# B&R Automation Studio project DuctLines (part 16)

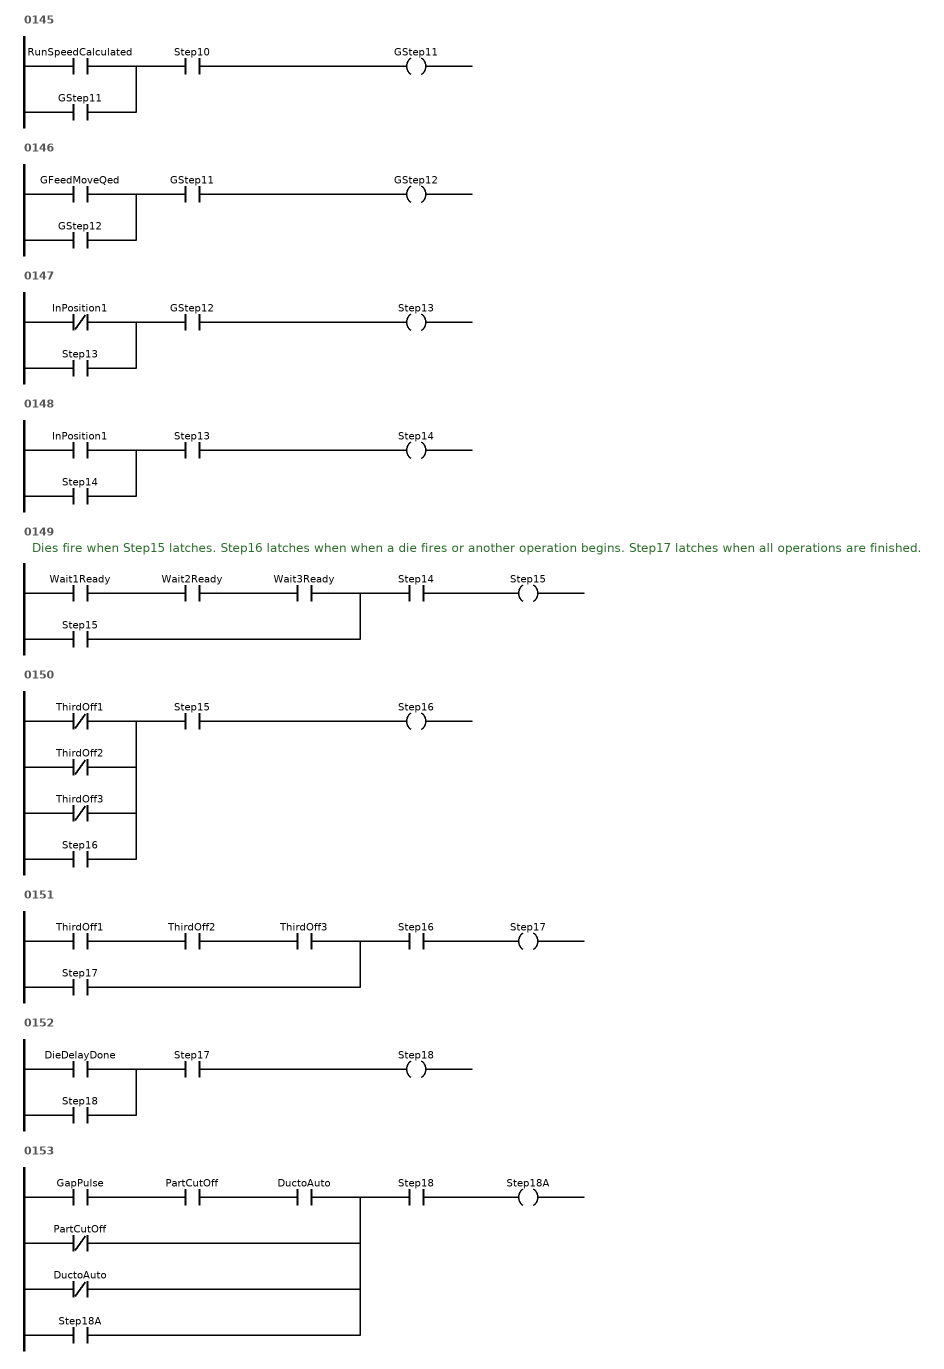
[picture p282: ladder Cyclic.ld]
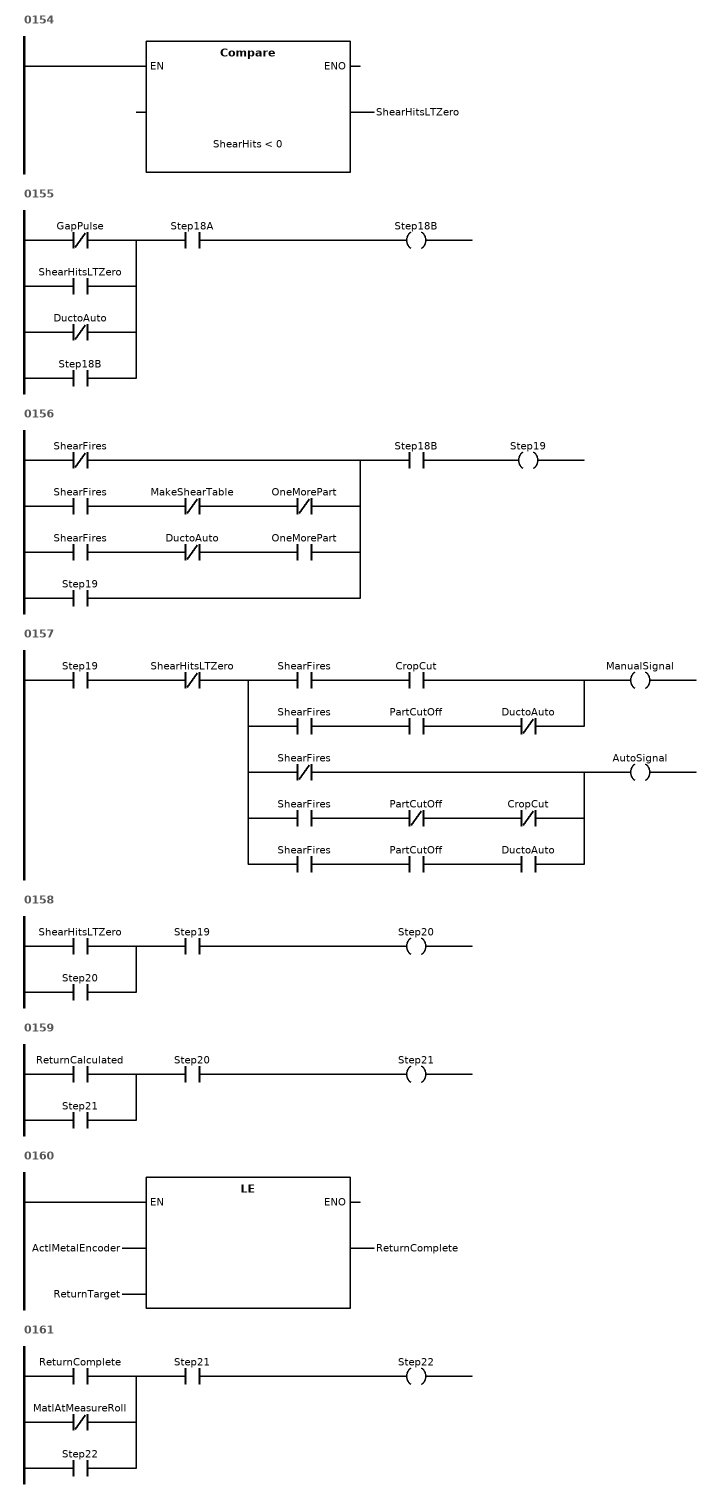
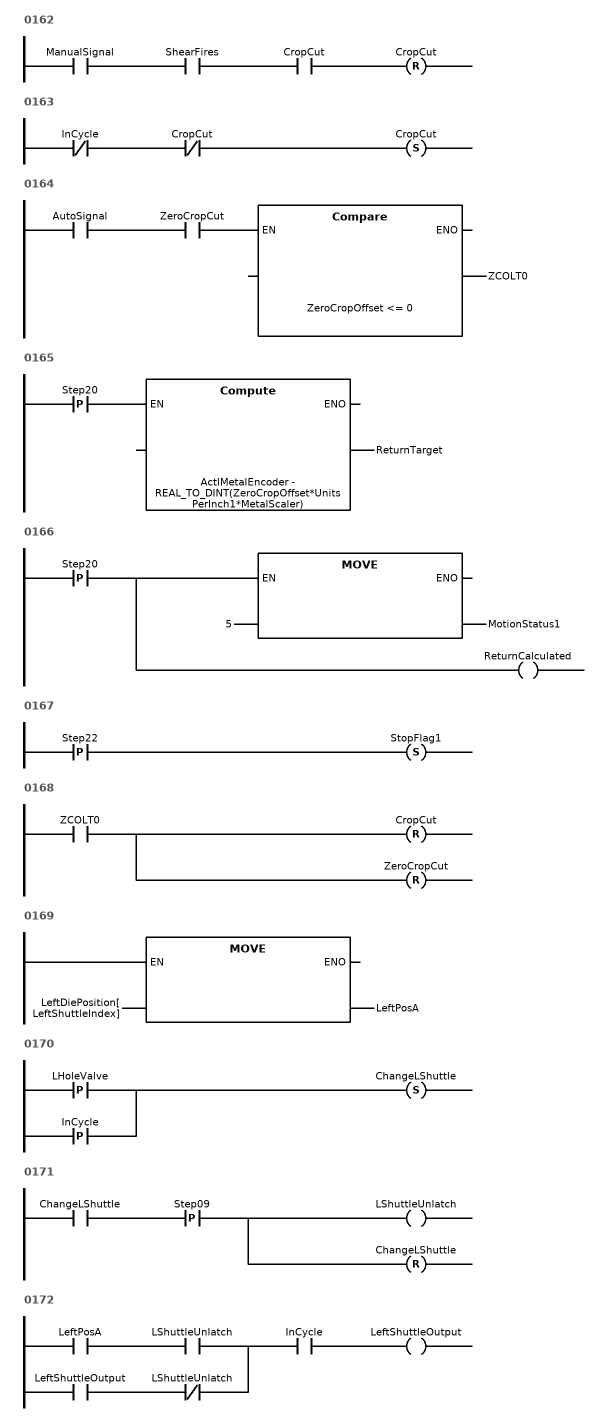
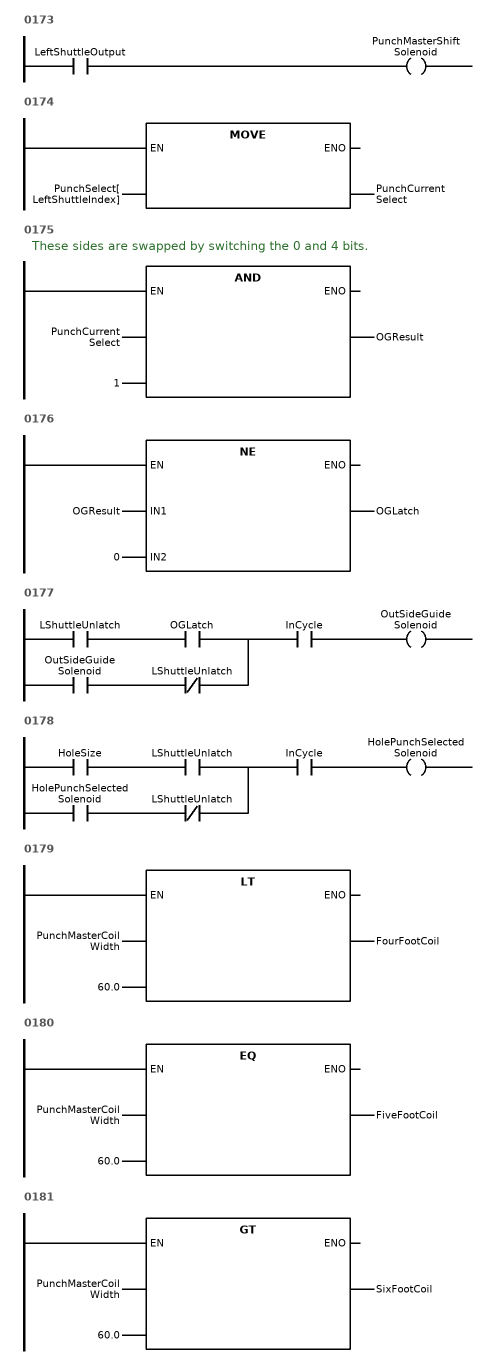
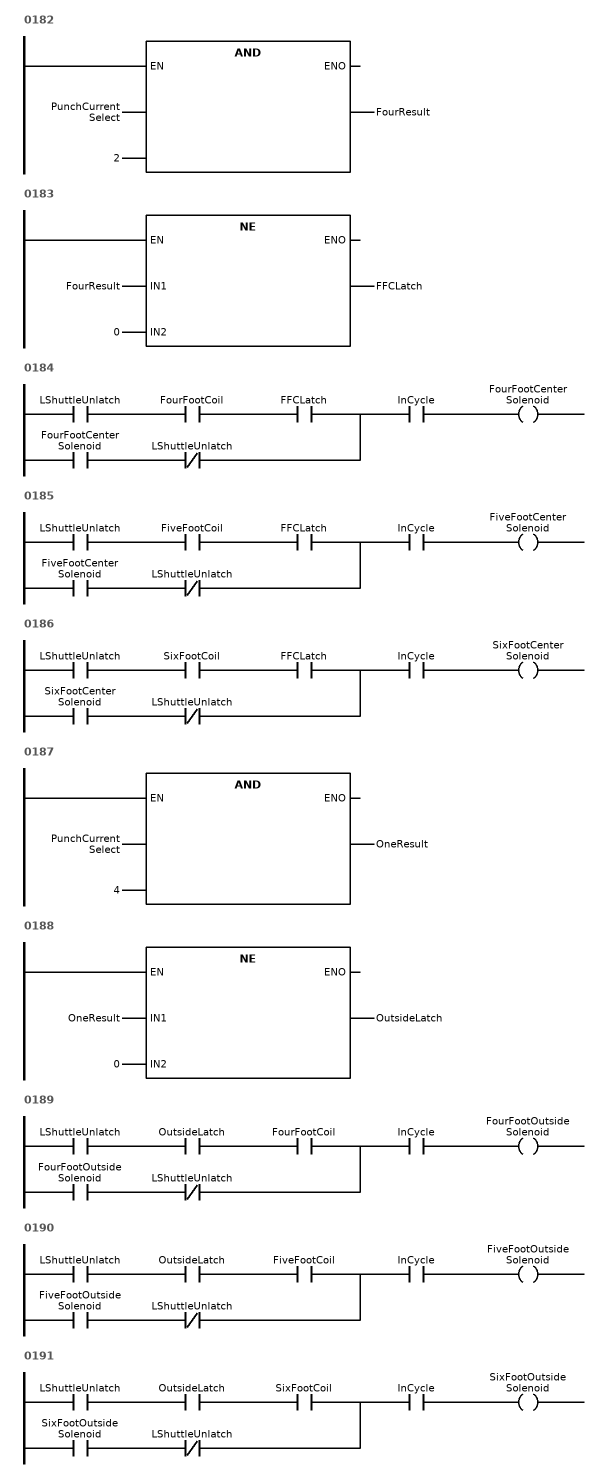
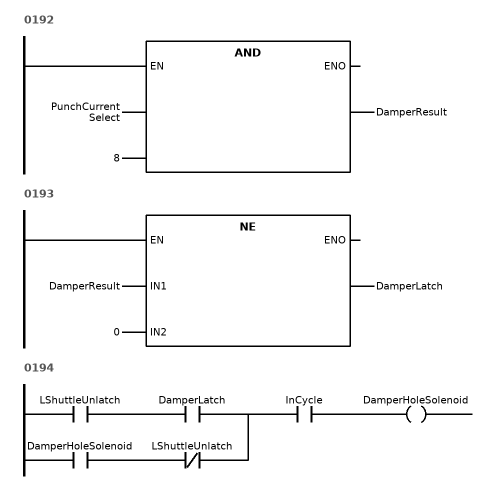
Ladder, written as Structured Text:
```iecst
PROGRAM _CYCLIC
VAR
    _e1 : R_TRIG;
    _e2 : R_TRIG;
    _e3 : R_TRIG;
    _e4 : F_TRIG;
    _e5 : F_TRIG;
    _e6 : R_TRIG;
    _e7 : R_TRIG;
    _e8 : R_TRIG;
    _e9 : R_TRIG;
    _e10 : R_TRIG;
    _e11 : F_TRIG;
    _e12 : F_TRIG;
    _e13 : F_TRIG;
    _e14 : R_TRIG;
    _e15 : R_TRIG;
    _e16 : R_TRIG;
    _e17 : R_TRIG;
    _e18 : R_TRIG;
    _e19 : R_TRIG;
    _e20 : R_TRIG;
    _e21 : R_TRIG;
    _e22 : R_TRIG;
    _e23 : R_TRIG;
    _e24 : R_TRIG;
    _e25 : R_TRIG;
    _e26 : F_TRIG;
    _e27 : R_TRIG;
    _e28 : R_TRIG;
    _e29 : F_TRIG;
    _e30 : R_TRIG;
    _e31 : R_TRIG;
    _e32 : R_TRIG;
    _e33 : R_TRIG;
    _e34 : F_TRIG;
    _e35 : R_TRIG;
    _e36 : F_TRIG;
    _e37 : R_TRIG;
    _e38 : F_TRIG;
    _e39 : R_TRIG;
    _e40 : F_TRIG;
    _e41 : R_TRIG;
    _e42 : F_TRIG;
    _e43 : R_TRIG;
    _e44 : F_TRIG;
    _e45 : R_TRIG;
    _e46 : F_TRIG;
    _e47 : R_TRIG;
    _e48 : F_TRIG;
    _e49 : R_TRIG;
    _e50 : F_TRIG;
    _e51 : R_TRIG;
    _e52 : F_TRIG;
    _e53 : R_TRIG;
    _e54 : F_TRIG;
    _e55 : R_TRIG;
    _e56 : R_TRIG;
    _e57 : R_TRIG;
    _e58 : R_TRIG;
    _e59 : R_TRIG;
    _e60 : F_TRIG;
    _e61 : R_TRIG;
    _e62 : R_TRIG;
    _e63 : F_TRIG;
    _e64 : R_TRIG;
    _e65 : R_TRIG;
    _p66 : BOOL;
    _e67 : R_TRIG;
    _e68 : R_TRIG;
    _e69 : R_TRIG;
    _e70 : R_TRIG;
    _p71 : BOOL;
    _e72 : F_TRIG;
    _e73 : R_TRIG;
    _e74 : R_TRIG;
    _e75 : R_TRIG;
    _e76 : R_TRIG;
    _e77 : R_TRIG;
    _e78 : R_TRIG;
    _e79 : R_TRIG;
    _e80 : R_TRIG;
END_VAR
(* Network 1: This routine doesn't handle a snap lock button gag. *)
MetalEncoder := ActlMetalEncoder - CoilAccumulator;

(* Network 2 *)
_e1(CLK := FSHydraulicsButton);
CLPUnlatch := _e1.Q AND CoilLinePower;

(* Network 3 *)
_e2(CLK := FSHydraulicsButton);
CoilLinePower := (_e2.Q OR CoilLinePower) AND AllSystemsOK AND NOT CLPUnlatch;

(* Network 4 *)
_e3(CLK := RollDriveEnableButton);
RollEnableUnlatch := _e3.Q AND ProcessorDriveEnable;

(* Network 5 *)
_e4(CLK := CoilLineHalt);
_e5(CLK := InCycle);
DuctoAutoUnlatch := (_e4.Q OR (Step18B AND NOT Step19) OR (Step18 AND OneMorePart) OR ManualSignal OR _e5.Q) AND DuctoAuto;

(* Network 6 *)
_e6(CLK := CoilLineRun);
DuctoAuto := (_e6.Q OR DuctoAuto) AND NOT DuctoAutoUnlatch;

(* Network 7 *)
CoilLineRunIndicator := DuctoAuto;

(* Network 8 *)
CoilLineHaltIndicator := NOT DuctoAuto;

(* Network 9: OneMorePart logic needs To Execute Before The FeedInitiate Signal rung. *)
JobChanging := (RunJob - 1)  <> ShearJob;

(* Network 10 *)
OneMorePart := (InCycle OR (OneMorePart AND NOT FeedInitiate)) AND JobChanging AND NOT RunContinuousSignal;

(* Network 11: Feed Initiate Signal *)
_e7(CLK := CoilLineRun);
FeedInitiate := _e7.Q AND AllSystemsOK AND ElectricServoStuffOK;

(* Network 12: Verify HMI Job change request *)
IF RunJobClick AND NOT InCycle THEN NewRunJobOk := NewRunJob <= MaxRunJob; END_IF;

(* Network 13 *)
IF RunJobClick AND NewRunJobOk AND NOT InCycle THEN RunJob := NewRunJob; END_IF;

(* Network 14 *)
IF RunJobClick THEN NewRunJobOk := FALSE; END_IF;

(* Network 15 *)
IF RunJobClick THEN RunJobClick := FALSE; END_IF;

(* Network 16: Update HMI job when the shear finishes one. *)
JobsDifferent := (RunJob - 1) <> ShearJob;

(* Network 17 *)
ChangeJob1 := InCycle AND Step19 AND ShearFires AND JobsDifferent;

(* Network 18 *)
IF ChangeJob1 THEN RunJob := ShearJob + 1; END_IF;

(* Network 19 *)
_e8(CLK := FeedInitiate);
IF _e8.Q THEN NoShearHits := FALSE; END_IF;

(* Network 20: Latch BatchActive in whenever the FeedInitiate signal comes on and the Ducto Sequence isn't started. Step04 latches after PC downloads tables and resets StartSignal. Unlatch BatchActive at that point if the shear has no hits. Step19 is the last one in the Ducto sequence. If there are no shear hits, the run is finished. BatchActive unlatches and the entire sequence unlatches. *)
SHLT0 := ShearHits < 0;

(* Network 21 *)
_e9(CLK := Step04);
NoShearHits := _e9.Q AND SHLT0;

(* Network 22 *)
_e10(CLK := WarningComplete);
_e11(CLK := MatlAtMeasureRoll);
_e12(CLK := EStopClear);
_e13(CLK := ProcessorDriveEnable);
BatchCancelUnlatch := CoilLineReset OR NoShearHits OR (_e10.Q AND NOT CoilLineRun) OR _e11.Q OR _e12.Q OR _e13.Q OR Step22;

(* Network 23 *)
InCycle := ((FeedInitiate AND NOT Step01) OR InCycle) AND NOT BatchCancelUnlatch;

(* Network 24: There are 3 of these timers *)
ZRCTon(IN := Step04A AND NOT Step04B, PT := T#500ms);
ZCReverseComplete := ZRCTon.Q;

(* Network 25 *)
DDDoneTimer(IN := Step04B AND NOT Step04C, PT := T#2s);
DirectionDelayDone := DDDoneTimer.Q;

(* Network 26 *)
ZCSCTimer(IN := Step04D, PT := T#2s);
ZCSettleComplete := ZCSCTimer.Q;

(* Network 27 *)
_e14(CLK := MatlAtMeasureRoll);
IF _e14.Q AND Step04C AND NOT Step04D THEN MetalEncoderLatch := ActlMetalEncoder; END_IF;

(* Network 28 *)
_e15(CLK := Step05A);
IF _e15.Q AND NOT ZeroCropCut THEN MetalEncoderLatch := ActlMetalEncoder; END_IF;

(* Network 29: First actions in Ducto sequence, reset indexes and moves, set start signal for PC to generate die tables. *)
IF Step01 AND NOT Step02 THEN
    ShearMove := 0.0;
    LTNotchMove := 0.0;
    VNotchMove := 0.0;
    LeftHoleMove := 0.0;
    CenterHoleMove := 0.0;
    RightHoleMove := 0.0;
    PartsMade := 0;
    ShearIndex := 0;
    LTNotchIndex := 0;
    VNotchIndex := 0;
    LeftHoleIndex := 0;
    CenterHoleIndex := 0;
    RightHoleIndex := 0;
    ButtonMove := 0.0;
    ShearBrakeMove := 0.0;
    CustomLTMove := 0.0;
    CleatMove := 0.0;
    ButtonIndex := 0;
    ShearBrakeIndex := 0;
    CustomLTIndex := 0;
END_IF;

(* Network 30 *)
IF Step01 AND NOT Step02 THEN
    CleatIndex := 0;
    ButtonActual := 0;
    CustomVMove := 0.0;
    CustomVIndex := 0;
    BeadRollMove := 0.0;
    BeadRollIndex := 0;
    StartSignal := TRUE;
END_IF;

(* Network 31: The Actual Material Counter Needs To Be Initialized To ZeroCropDifference Here, too. *)
_e16(CLK := Step05A);
IF _e16.Q THEN
    ZeroCropDifference := MetalEncoderLatch - ActlMetalEncoder;
    CoilAccumulator := ZeroCropDifference;
    MetalTarget := ZeroCropDifference;
END_IF;

(* Network 32 *)
TON_1(IN := Step05A, PT := T#200ms);
PartRefOK := TON_1.Q;

(* Network 33 *)
ProcessorEncoderReset := (Step05A AND NOT Step05B) OR (ShearValve AND NOT InCycle);

(* Network 34 *)
TON_Warning(IN := Step02 AND NOT Step03, PT := WarningDelay1);
WarningComplete := TON_Warning.Q;

(* Network 35 *)
WarningHorn := Step02 AND NOT Step03;

(* Network 36: Reset variable to get ready for a new move *)
IF Step06 AND NOT Step07 THEN
    PartCutOff := FALSE;
    ShearFires := FALSE;
    IncrementalRealTarget := 0.0;
END_IF;
InitMoveSignal := Step06 AND NOT Step07;

(* Network 37: Make Sure All Data Is Updated By PC *)
HalfUpdated1 := NOT MakeShearTable AND NOT MakeLTTable AND NOT MakeVTable AND NOT MakeLHoleTable AND NOT MakeCHoleTable;

(* Network 38 *)
HalfUpdated2 := NOT MakeRHoleTable AND NOT MakeButtonTable AND NOT MakeShearBrakeTable AND NOT MakeCleatTable;

(* Network 39 *)
DataUpdated := HalfUpdated1 AND HalfUpdated2;

(* Network 40: New Connector Logic *)
_e17(CLK := Step04);
IF _e17.Q THEN SavedConnector := LatestConnector; END_IF;

(* Network 41 *)
_e18(CLK := Step08);
IF _e18.Q THEN SetConnectorChange := (LatestConnector <> SavedConnector) AND (LTNotchHits > 0); END_IF;

(* Network 42 *)
ChangeConnector := SetConnectorChange OR (ChangeConnector AND NOT LTValve AND InCycle);

(* Network 43: Net #37-40 from PicPro.  *)
MUX1:
_e19(CLK := Step08);
IF _e19.Q AND ShearUsedUp THEN
    ShearMove := MUX(K := ShearIndex, IN2 := ShearTable[0], IN3 := ShearTable[1], IN4 := ShearTable[2], IN5 := ShearTable[3], IN6 := ShearTable[4], IN7 := ShearTable[5]);
END_IF;
IF _e19.Q AND LTUsedUp THEN
    LTNotchMove := MUX(K := LTNotchIndex, IN2 := LTNotchTable[0], IN3 := LTNotchTable[1], IN4 := LTNotchTable[2], IN5 := LTNotchTable[3], IN6 := LTNotchTable[4], IN7 := LTNotchTable[5]);
END_IF;
IF _e19.Q AND VUsedUp THEN
    VNotchMove := MUX(K := VNotchIndex, IN2 := VNotchTable[0], IN3 := VNotchTable[1], IN4 := VNotchTable[2], IN5 := VNotchTable[3], IN6 := VNotchTable[4], IN7 := VNotchTable[5]);
END_IF;

(* Network 44 *)
_e20(CLK := Step08);
IF _e20.Q AND ButtonUsedUp THEN
    ButtonMove := MUX(K := ButtonIndex, IN2 := ButtonTable[0], IN3 := ButtonTable[1], IN4 := ButtonTable[2], IN5 := ButtonTable[3], IN6 := ButtonTable[4], IN7 := ButtonTable[5]);
END_IF;
IF _e20.Q AND ShearBrakeUsedUp THEN
    ShearBrakeMove := MUX(K := ShearBrakeIndex, IN2 := ShearBrakeTable[0], IN3 := ShearBrakeTable[1], IN4 := ShearBrakeTable[2], IN5 := ShearBrakeTable[3], IN6 := ShearBrakeTable[4], IN7 := ShearBrakeTable[5]);
END_IF;
IF _e20.Q AND CustomLTUsedUp THEN
    CustomLTMove := MUX(K := CustomLTIndex, IN2 := CustomLTTable[0], IN3 := CustomLTTable[1], IN4 := CustomLTTable[2], IN5 := CustomLTTable[3], IN6 := CustomLTTable[4], IN7 := CustomLTTable[5]);
END_IF;

(* Network 45 *)
_e21(CLK := Step08);
IF _e21.Q AND CleatUsedUp THEN
    CleatMove := MUX(K := CleatIndex, IN2 := CleatTable[0], IN3 := CleatTable[1], IN4 := CleatTable[2], IN5 := CleatTable[3], IN6 := CleatTable[4], IN7 := CleatTable[5]);
END_IF;
IF _e21.Q AND CustomVUsedUp THEN
    CustomVMove := MUX(K := CustomVIndex, IN2 := CustomVTable[0], IN3 := CustomVTable[1], IN4 := CustomVTable[2], IN5 := CustomVTable[3], IN6 := CustomVTable[4], IN7 := CustomVTable[5]);
END_IF;

(* Network 46: These 4 tables have too many values for the B&R mux. *)
_e22(CLK := Step08);
IF _e22.Q AND LeftHoleUsedUp THEN LeftHoleMove := LeftHoleTable[LeftHoleIndex]; END_IF;
IF _e22.Q AND CenterHoleUsedUp THEN CenterHoleMove := CenterHoleTable[CenterHoleIndex]; END_IF;
IF _e22.Q AND RightHoleUsedUp THEN RightHoleMove := RightHoleTable[RightHoleIndex]; END_IF;
IF _e22.Q AND BeadRollUsedUp THEN BeadRollMove := BeadRollTable[BeadRollIndex]; END_IF;

(* Network 47 *)
_e23(CLK := Step08);
IF _e23.Q THEN
    LeftShuttleIndex := LeftHoleIndex;
    CenterShuttleIndex := CenterHoleIndex;
    RightShuttleIndex := RightHoleIndex;
END_IF;

(* Network 48 *)
_e24(CLK := Step08);
IF _e24.Q THEN getNextMove; END_IF;

(* Network 49 *)
_e25(CLK := Step08A);
_e26(CLK := InCycle);
IF _e25.Q OR _e26.Q THEN NextMoveDone := FALSE; END_IF;

(* Network 50 *)
ShearUsedUp := ABS(ShearMove) <= InPositionBand;

(* Network 51 *)
LTUsedUp := ABS(LTNotchMove) <= InPositionBand;

(* Network 52 *)
VUsedUp := ABS(VNotchMove) <= InPositionBand;

(* Network 53 *)
LeftHoleUsedUp := ABS(LeftHoleMove) <= InPositionBand;

(* Network 54 *)
CenterHoleUsedUp := ABS(CenterHoleMove) <= InPositionBand;

(* Network 55 *)
RightHoleUsedUp := ABS(RightHoleMove) <= InPositionBand;

(* Network 56 *)
ButtonUsedUp := ABS(ButtonMove) <= InPositionBand;

(* Network 57 *)
ShearBrakeUsedUp := ABS(ShearBrakeMove) <= InPositionBand;

(* Network 58 *)
CustomLTUsedUp := ABS(CustomLTMove) <= InPositionBand;

(* Network 59 *)
CleatUsedUp := ABS(CleatMove) <= InPositionBand;

(* Network 60 *)
CustomVUsedUp := ABS(CustomVMove) <= InPositionBand;

(* Network 61 *)
BeadRollUsedUp := ABS(BeadRollMove) <= InPositionBand;

(* Network 62 *)
_e27(CLK := Step08A);
IF _e27.Q THEN UpdateTables; END_IF;

(* Network 63 *)
_e28(CLK := Step08B);
_e29(CLK := InCycle);
IF _e28.Q OR _e29.Q THEN UpdateTablesDone := FALSE; END_IF;

(* Network 64 *)
_e30(CLK := Step08B);
IF _e30.Q THEN IncrementalRealTarget := IncrementalRealTarget + SmallResult; END_IF;

(* Network 65 *)
_e31(CLK := Step08B);
NextMoveComplete := _e31.Q AND (ShearFires OR LTFires OR VFires OR LeftHoleFires OR CenterHoleFires OR RightHoleFires OR ButtonFires OR ShearBrakeFires OR CustomLTFires OR CleatFires OR CustomVFires OR BeadRollFires);

(* Network 66 *)
_e32(CLK := Step08B);
NextMoveLookAgain := _e32.Q AND NOT NextMoveComplete;

(* Network 67 *)
_e33(CLK := LTValve);
_e34(CLK := InCycle);
IF _e33.Q OR _e34.Q THEN LTFires := FALSE; END_IF;

(* Network 68 *)
_e35(CLK := VValve);
_e36(CLK := InCycle);
IF _e35.Q OR _e36.Q THEN VFires := FALSE; END_IF;

(* Network 69 *)
_e37(CLK := LHoleValve);
_e38(CLK := InCycle);
IF _e37.Q OR _e38.Q THEN LeftHoleFires := FALSE; END_IF;

(* Network 70 *)
_e39(CLK := CHoleValve);
_e40(CLK := InCycle);
IF _e39.Q OR _e40.Q THEN CenterHoleFires := FALSE; END_IF;

(* Network 71 *)
_e41(CLK := RHoleValve);
_e42(CLK := InCycle);
IF _e41.Q OR _e42.Q THEN RightHoleFires := FALSE; END_IF;

(* Network 72 *)
_e43(CLK := CycleButtons);
_e44(CLK := InCycle);
IF _e43.Q OR _e44.Q THEN ButtonFires := FALSE; END_IF;

(* Network 73 *)
_e45(CLK := CycleMaleBender);
_e46(CLK := InCycle);
IF _e45.Q OR _e46.Q THEN ShearBrakeFires := FALSE; END_IF;

(* Network 74 *)
_e47(CLK := CustomLTValve);
_e48(CLK := InCycle);
IF _e47.Q OR _e48.Q THEN CustomLTFires := FALSE; END_IF;

(* Network 75 *)
_e49(CLK := ChangeKDRolls);
_e50(CLK := InCycle);
IF _e49.Q OR _e50.Q THEN CleatFires := FALSE; END_IF;

(* Network 76 *)
_e51(CLK := CustomVValve);
_e52(CLK := InCycle);
IF _e51.Q OR _e52.Q THEN CustomVFires := FALSE; END_IF;

(* Network 77 *)
_e53(CLK := WaitCon3);
_e54(CLK := InCycle);
IF _e53.Q OR _e54.Q THEN BeadRollFires := FALSE; END_IF;

(* Network 78 *)
_e55(CLK := Step09);
IF _e55.Q THEN MetalScaler := MetalDesired / MetalActual; END_IF;
ClearEncoderSignal := _e55.Q;

(* Network 79: This doesn't hurt anything when the 2 speed hydraulic feed system is used. *)
_e56(CLK := Step10);
IF _e56.Q AND CropCut THEN RunSpeed1 := CropPercent1; END_IF;
IF _e56.Q AND NOT CropCut THEN RunSpeed1 := PercentSpeed1; END_IF;
RunSpeedCalculated := _e56.Q;

(* Network 80 *)
WaitToFire1 := Step14 AND LTFires AND ChangeConnector;
WaitCon1 := Step14 AND FeedInitiate;

(* Network 81 *)
TON_10(IN := WaitToFire2, PT := T#50ms);
WaitCon2 := TON_10.Q;

(* Network 82 *)
_e57(CLK := InPosition1);
WaitToFire2 := (_e57.Q OR WaitToFire2) AND NOT WaitCon2;

(* Network 83 *)
WaitCon3 := Step14 AND BeadRollFires AND FeedInitiate;
WaitToFire3 := Step14 AND BeadRollFires;

(* Network 84 *)
_e58(CLK := WaitToFire3);
IF _e58.Q THEN ChangeBeadRoll := TRUE; END_IF;

(* Network 85 *)
Wait1Ready := Step14 AND ((WaitToFire1 AND WaitCon1) OR NOT WaitToFire1);
Wait2Ready := Step14 AND ((WaitToFire2 AND WaitCon2) OR NOT WaitToFire2);
Wait3Ready := Step14 AND ((WaitToFire3 AND WaitCon3) OR NOT WaitToFire3);

(* Network 86 *)
IF (Step15 AND ShearFires) OR (NOT InCycle AND CycleShear) THEN
    shearTime := DINT_TO_TIME(ShearDwell);
END_IF;

(* Network 87 *)
TP_0(IN := (Step15 AND ShearFires) OR (NOT InCycle AND CycleShear), PT := shearTime);
ShearValve := TP_0.Q;

(* Network 88 *)
IF CycleShear THEN CycleShear := FALSE; END_IF;

(* Network 89 *)
IF (Step15 AND LTFires) OR (NOT InCycle AND CycleLTDie) THEN LTTime := DINT_TO_TIME(LTDwell); END_IF;

(* Network 90 *)
TP_1(IN := (Step15 AND LTFires) OR (NOT InCycle AND CycleLTDie), PT := LTTime);
LTValve := TP_1.Q;

(* Network 91 *)
IF CycleLTDie THEN CycleLTDie := FALSE; END_IF;

(* Network 92 *)
IF (Step15 AND VFires) OR (NOT InCycle AND CycleVDie) THEN VTime := DINT_TO_TIME(VDwell); END_IF;

(* Network 93 *)
TP_2(IN := (Step15 AND VFires) OR (NOT InCycle AND CycleVDie), PT := VTime);
VValve := TP_2.Q;

(* Network 94 *)
IF CycleVDie THEN CycleVDie := FALSE; END_IF;

(* Network 95 *)
IF (Step15 AND LeftHoleFires) OR (NOT InCycle AND CycleLDie) THEN
    LeftHoleTime := DINT_TO_TIME(LHoleDwell);
END_IF;

(* Network 96 *)
TP_3(IN := (Step15 AND LeftHoleFires) OR (NOT InCycle AND CycleLDie), PT := LeftHoleTime);
LHoleValve := TP_3.Q;

(* Network 97 *)
IF CycleLDie THEN CycleLDie := FALSE; END_IF;

(* Network 98 *)
IF (Step15 AND CenterHoleFires) OR (NOT InCycle AND CycleCDie) THEN
    CenterHoleTime := DINT_TO_TIME(CHoleDwell);
END_IF;

(* Network 99 *)
TP_4(IN := (Step15 AND CenterHoleFires) OR (NOT InCycle AND CycleCDie), PT := CenterHoleTime);
CHoleValve := TP_4.Q;

(* Network 100 *)
IF (Step15 AND RightHoleFires) OR (NOT InCycle AND CycleRDie) THEN
    RightHoleTime := DINT_TO_TIME(RHoleDwell);
END_IF;

(* Network 101 *)
TP_5(IN := (Step15 AND RightHoleFires) OR (NOT InCycle AND CycleRDie), PT := RightHoleTime);
RHoleValve := TP_5.Q;

(* Network 102 *)
IF (Step15 AND CustomLTFires) OR (NOT InCycle AND CycleCustomLTDie) THEN
    CustomLTTime := DINT_TO_TIME(CustomLTDwell);
END_IF;

(* Network 103 *)
TP_6(IN := (Step15 AND CustomLTFires) OR (NOT InCycle AND CycleCustomLTDie), PT := CustomLTTime);
CustomLTValve := TP_6.Q;

(* Network 104 *)
IF (Step15 AND CustomVFires) OR (NOT InCycle AND CycleCustomVDie) THEN
    CustomVTime := DINT_TO_TIME(CustomVDwell);
END_IF;

(* Network 105 *)
TP_7(IN := (Step15 AND CustomVFires) OR (NOT InCycle AND CycleCustomVDie), PT := CustomVTime);
CustomVValve := TP_7.Q;

(* Network 106 *)
_e59(CLK := ButtonBack7);
_e60(CLK := InCycle);
UnlatchButtons := (Step15 AND _e59.Q) OR _e60.Q;

(* Network 107 *)
_e61(CLK := Step15);
CycleButtons := ((_e61.Q AND ButtonFires) OR CycleButtons) AND NOT UnlatchButtons;

(* Network 108 *)
_e62(CLK := ShearClampUpProx);
_e63(CLK := ProcessorDriveEnable);
UnlatchBender := ((Step15 OR ShearBrakeLatch) AND _e62.Q) OR _e63.Q;

(* Network 109 *)
IF UnlatchBender THEN ShearBrakeLatch := FALSE; END_IF;

(* Network 110 *)
_e64(CLK := Step15);
CycleMaleBender := ((_e64.Q AND ShearBrakeFires) OR ShearBrakeLatch OR CycleMaleBender) AND NOT UnlatchBender;

(* Network 111 *)
_e65(CLK := Step15);
ChangeKDRolls := _e65.Q AND CleatFires;

(* Network 112 *)
LeftKnockDownRoll := (ChangeKDRolls AND LeftCleatEnable AND NOT LeftKnockDownRoll) OR (LeftKnockDownRoll AND InCycle AND NOT ChangeKDRolls);

(* Network 113 *)
RightKnockDownRoll := (ChangeKDRolls AND RightCleatEnable AND NOT RightKnockDownRoll) OR (RightKnockDownRoll AND InCycle AND NOT ChangeKDRolls);

(* Network 114 *)
_p66 := NOT ShearValve AND NOT LTValve AND NOT VValve AND NOT LHoleValve;
ThirdOff1 := _p66 AND (HolePunchUp OR NOT PunchMaster);

(* Network 115 *)
ThirdOff2 := NOT CHoleValve AND NOT RHoleValve AND NOT ChangeKDRolls AND NOT CycleMaleBender;

(* Network 116 *)
ThirdOff3 := NOT CycleButtons AND NOT CustomLTValve AND NOT CustomVValve AND NOT WaitCon3;

(* Network 117 *)
_e67(CLK := Step17);
IF _e67.Q THEN DieUpTime := DINT_TO_TIME(DieUpDelay); END_IF;

(* Network 118 *)
TON_0(IN := Step17 AND NOT Step18, PT := DieUpTime);
DieDelayDone := TON_0.Q;

(* Network 119 *)
IncPartsMade := PartCutOff;

(* Network 120 *)
_e68(CLK := Step18);
IF _e68.Q THEN GTime := DINT_TO_TIME(GapTime); END_IF;

(* Network 121 *)
TP_8(IN := Step18 AND PartCutOff AND DuctoAuto, PT := GTime);
GapTP := TP_8.Q;

(* Network 122 *)
_e69(CLK := Step18);
GapPulse := GapTP OR _e69.Q;

(* Network 123 *)
_e70(CLK := Step18);
IF _e70.Q AND IncPartsMade THEN
    PartsMade := PartsMade + 1;
    RTotalInches := PartLength + RTotalInches;
END_IF;

(* Network 124 *)
IF ChangeJob1 THEN PartsMade := 0; END_IF;

(* Network 125 *)
TotalInches := RTotalInches;

(* Network 126 *)
IF ClearLengthCountSignal THEN RTotalInches := 0; END_IF;
_p71 := ClearLengthCountSignal;
IF _p71 THEN ClearLengthCountSignal := FALSE; END_IF;

(* Network 127: Set StartSignal for touchscreen. Do the warning while waiting for data. Touchscreen resets StartSignal at the tail end of the data transfer. *)
Step01 := (FeedInitiate OR Step01) AND InCycle;

(* Network 128 *)
Step02 := (StartSignal OR Step02) AND Step01;

(* Network 129 *)
Step03 := (WarningComplete OR Step03) AND Step02;

(* Network 130 *)
Step04 := (NOT StartSignal OR Step04) AND Step03;

(* Network 131: Position material for no crop cut. Latch these rungs in if crop cutting. *)
_e72(CLK := MatlAtMeasureRoll);
Step04A := (_e72.Q OR NOT ZeroCropCut OR Step04A) AND Step04;

(* Network 132 *)
Step04B := (ZCReverseComplete OR NOT ZeroCropCut OR Step04B) AND Step04A;

(* Network 133 *)
Step04C := (DirectionDelayDone OR NOT ZeroCropCut OR Step04C) AND Step04B;

(* Network 134 *)
_e73(CLK := MatlAtMeasureRoll);
Step04D := (_e73.Q OR NOT ZeroCropCut OR Step04D) AND Step04C;

(* Network 135 *)
Step04E := (ZCSettleComplete OR Step04E) AND Step04D;

(* Network 136 *)
Step05A := (ServoLoop1Closed OR Step05A) AND Step04E;

(* Network 137 *)
Step05B := (PartRefOK OR Step05B) AND Step05A;

(* Network 138: The last step in the sequence determines if the processor should stop to wait for the FeedInitiate signal. The manual signal is set if the processor needs to stop. The manual signal ujnlatches all steps past Step05B and the waits at Step05B for for FeedInitiate. The auto signal is set if the processor can continue without a FeedInitiate signal. The auto signal unlatches all steps past Step06. *)
_e74(CLK := Step05B);
Step06 := (FeedInitiate OR _e74.Q OR Step06) AND Step05B AND NOT ManualSignal;

(* Network 139 *)
Step07 := (InitMoveSignal OR Step07) AND Step06 AND NOT AutoSignal;

(* Network 140: Step08 enables the the rungs that determine the length of the next move and what to do when it completes. This will execute multiple times in some cases before it is finished. *)
Step08 := (DataUpdated OR Step08) AND Step07 AND NOT NextMoveLookAgain;

(* Network 141 *)
Step08A := (NextMoveDone OR Step08A) AND Step08;

(* Network 142 *)
Step08B := (UpdateTablesDone OR Step08B) AND Step08A;

(* Network 143 *)
Step09 := (NextMoveComplete OR Step09) AND Step08B;

(* Network 144 *)
Step10 := (ClearEncoderSignal OR Step10) AND Step09;

(* Network 145 *)
GStep11 := (RunSpeedCalculated OR GStep11) AND Step10;

(* Network 146 *)
GStep12 := (GFeedMoveQed OR GStep12) AND GStep11;

(* Network 147 *)
Step13 := (NOT InPosition1 OR Step13) AND GStep12;

(* Network 148 *)
Step14 := (InPosition1 OR Step14) AND Step13;

(* Network 149: Dies fire when Step15 latches. Step16 latches when when a die fires or another operation begins. Step17 latches when all operations are finished. *)
Step15 := ((Wait1Ready AND Wait2Ready AND Wait3Ready) OR Step15) AND Step14;

(* Network 150 *)
Step16 := (NOT ThirdOff1 OR NOT ThirdOff2 OR NOT ThirdOff3 OR Step16) AND Step15;

(* Network 151 *)
Step17 := ((ThirdOff1 AND ThirdOff2 AND ThirdOff3) OR Step17) AND Step16;

(* Network 152 *)
Step18 := (DieDelayDone OR Step18) AND Step17;

(* Network 153 *)
Step18A := ((GapPulse AND PartCutOff AND DuctoAuto) OR NOT PartCutOff OR NOT DuctoAuto OR Step18A) AND Step18;

(* Network 154 *)
ShearHitsLTZero := ShearHits < 0;

(* Network 155 *)
Step18B := (NOT GapPulse OR ShearHitsLTZero OR NOT DuctoAuto OR Step18B) AND Step18A;

(* Network 156 *)
Step19 := (NOT ShearFires OR (ShearFires AND ((NOT MakeShearTable AND NOT OneMorePart) OR (NOT DuctoAuto AND OneMorePart))) OR Step19) AND Step18B;

(* Network 157 *)
ManualSignal := Step19 AND NOT ShearHitsLTZero AND ShearFires AND (CropCut OR (PartCutOff AND NOT DuctoAuto));
AutoSignal := Step19 AND NOT ShearHitsLTZero AND (NOT ShearFires OR (ShearFires AND ((NOT PartCutOff AND NOT CropCut) OR (PartCutOff AND DuctoAuto))));

(* Network 158 *)
Step20 := (ShearHitsLTZero OR Step20) AND Step19;

(* Network 159 *)
Step21 := (ReturnCalculated OR Step21) AND Step20;

(* Network 160 *)
ReturnComplete := ActlMetalEncoder <= ReturnTarget;

(* Network 161 *)
Step22 := (ReturnComplete OR NOT MatlAtMeasureRoll OR Step22) AND Step21;

(* Network 162 *)
IF ManualSignal AND ShearFires AND CropCut THEN CropCut := FALSE; END_IF;

(* Network 163 *)
IF NOT InCycle AND NOT CropCut THEN CropCut := TRUE; END_IF;

(* Network 164 *)
IF AutoSignal AND ZeroCropCut THEN ZCOLT0 := ZeroCropOffset <= 0; END_IF;

(* Network 165 *)
_e75(CLK := Step20);
IF _e75.Q THEN
    ReturnTarget := ActlMetalEncoder - REAL_TO_DINT(ZeroCropOffset*UnitsPerInch1*MetalScaler);
END_IF;

(* Network 166 *)
_e76(CLK := Step20);
IF _e76.Q THEN MotionStatus1 := 5; END_IF;
ReturnCalculated := _e76.Q;

(* Network 167 *)
_e77(CLK := Step22);
IF _e77.Q THEN StopFlag1 := TRUE; END_IF;

(* Network 168 *)
IF ZCOLT0 THEN
    CropCut := FALSE;
    ZeroCropCut := FALSE;
END_IF;

(* Network 169 *)
LeftPosA := LeftDiePosition[LeftShuttleIndex];

(* Network 170 *)
_e78(CLK := LHoleValve);
_e79(CLK := InCycle);
IF _e78.Q OR _e79.Q THEN ChangeLShuttle := TRUE; END_IF;

(* Network 171 *)
_e80(CLK := Step09);
LShuttleUnlatch := ChangeLShuttle AND _e80.Q;
IF ChangeLShuttle AND _e80.Q THEN ChangeLShuttle := FALSE; END_IF;

(* Network 172 *)
LeftShuttleOutput := ((LeftPosA AND LShuttleUnlatch) OR (LeftShuttleOutput AND NOT LShuttleUnlatch)) AND InCycle;

(* Network 173 *)
PunchMasterShiftSolenoid := LeftShuttleOutput;

(* Network 174 *)
PunchCurrentSelect := PunchSelect[LeftShuttleIndex];

(* Network 175: These sides are swapped by switching the 0 and 4 bits. *)
OGResult := PunchCurrentSelect AND 1;

(* Network 176 *)
OGLatch := OGResult <> 0;

(* Network 177 *)
OutSideGuideSolenoid := ((LShuttleUnlatch AND OGLatch) OR (OutSideGuideSolenoid AND NOT LShuttleUnlatch)) AND InCycle;

(* Network 178 *)
HolePunchSelectedSolenoid := ((HoleSize AND LShuttleUnlatch) OR (HolePunchSelectedSolenoid AND NOT LShuttleUnlatch)) AND InCycle;

(* Network 179 *)
FourFootCoil := PunchMasterCoilWidth < 60.0;

(* Network 180 *)
FiveFootCoil := PunchMasterCoilWidth = 60.0;

(* Network 181 *)
SixFootCoil := PunchMasterCoilWidth > 60.0;

(* Network 182 *)
FourResult := PunchCurrentSelect AND 2;

(* Network 183 *)
FFCLatch := FourResult <> 0;

(* Network 184 *)
FourFootCenterSolenoid := ((LShuttleUnlatch AND FourFootCoil AND FFCLatch) OR (FourFootCenterSolenoid AND NOT LShuttleUnlatch)) AND InCycle;

(* Network 185 *)
FiveFootCenterSolenoid := ((LShuttleUnlatch AND FiveFootCoil AND FFCLatch) OR (FiveFootCenterSolenoid AND NOT LShuttleUnlatch)) AND InCycle;

(* Network 186 *)
SixFootCenterSolenoid := ((LShuttleUnlatch AND SixFootCoil AND FFCLatch) OR (SixFootCenterSolenoid AND NOT LShuttleUnlatch)) AND InCycle;

(* Network 187 *)
OneResult := PunchCurrentSelect AND 4;

(* Network 188 *)
OutsideLatch := OneResult <> 0;

(* Network 189 *)
FourFootOutsideSolenoid := ((LShuttleUnlatch AND OutsideLatch AND FourFootCoil) OR (FourFootOutsideSolenoid AND NOT LShuttleUnlatch)) AND InCycle;

(* Network 190 *)
FiveFootOutsideSolenoid := ((LShuttleUnlatch AND OutsideLatch AND FiveFootCoil) OR (FiveFootOutsideSolenoid AND NOT LShuttleUnlatch)) AND InCycle;

(* Network 191 *)
SixFootOutsideSolenoid := ((LShuttleUnlatch AND OutsideLatch AND SixFootCoil) OR (SixFootOutsideSolenoid AND NOT LShuttleUnlatch)) AND InCycle;

(* Network 192 *)
DamperResult := PunchCurrentSelect AND 8;

(* Network 193 *)
DamperLatch := DamperResult <> 0;

(* Network 194 *)
DamperHoleSolenoid := ((LShuttleUnlatch AND DamperLatch) OR (DamperHoleSolenoid AND NOT LShuttleUnlatch)) AND InCycle;
END_PROGRAM
```

Listed in the project but not available here: Logical/Global.typ, Logical/Libraries/MestekLib/Types.typ, Logical/Libraries/MestekLib/Constants.var, Logical/Feeder/Init.ld, Logical/Feeder/Exit.ld, Logical/Feeder/Types.typ, Logical/LibAsTCP1_ST/LibAsTCP1_ST.var, Logical/LibAsTCP1_ST/Client/Client.typ, Logical/LibAsTCP1_ST/Library/Types.typ, Logical/LibAsTCP1_ST/Library/Constants.var, Logical/LibAsTCP1_ST/Library/Library.fun, Logical/SBrake/Init.ld, Logical/SBrake/Exit.ld, Logical/SBrake/Types.typ, Logical/Uncoiler_2/Exit.ld, Logical/Uncoiler_2/Types.typ, Logical/IMotion1/Init.st, Logical/IMotion1/Exit.st, Logical/IMotion1/Types.typ
